(*
  Mark camera system on WEU machine
  1 mark sensor (optional: reverse mode - roll printed in reversed direction, sensor moved to other side)
*)
FUNCTION_BLOCK FB_MarkCamera_WEU EXTENDS FB_CameraBase
VAR_INPUT
  bReadyForPrinting             : BOOL;     // 
  nCurrentPosition              : DINT;     // current print postion
  fCurrentSpeed                 : LREAL;    // current print speed
  bPrintMarkExist               : BOOL;     // [from machine] print mark existing
  bPrintDirReverse              : BOOL;     // [from machine] print substrate in reverse direction
  nUsePerRepeatInLine           : UDINT;    // [from machine] use per repeat
  fMarkSizeDefault              : LREAL;    // mark size "a" [m]
  fMarkDistRepeatToStartMark    : LREAL;    // mark distance from repeat to start mark [m]
  fMarkDistFromCenter           : LREAL;    // mark distance from center [m]
END_VAR
VAR
  fbMarkDefinition   : FB_MarkDefinition;   // mark definition instance (used by MarkDetection)
  fbMarkDetection    : FB_MarkDetection;    // StartPosTrigger, CameraTrigger and MarkDetection (Mark handler for MarkCamera)
  
  // teach info
  _bTeachOk                     : BOOL;
  _nTeachedPoints               : UDINT;
  _nDetectedMarks               : UDINT;
  
  // status
  _bTeachError                  : BOOL;     // teach was not successful
  _bImageLengthError            : BOOL;     // invalid image/repeat length
  _bMarkDefinitionError         : BOOL;     // invalid mark definition
END_VAR
VAR CONSTANT
  fC_MinImageLength : LREAL := 0.05;  // minimal "repeat" length
END_VAR
VAR PERSISTENT
  eMarkMode     : E_MarkMode := E_MarkMode.AutoDefault;   // mark generation/detection mode
  bMarkInverted : BOOL;             // mark triangle are flipped on x axis
  nUsePerRepeat : UDINT := 4;       // number of "use" per repeat
  fMarkSpec_a   : LREAL := 0.005;   // mark spec a [m] - mark width
  fMarkSpec_b   : LREAL := 0.005;   // mark spec b [m] - (optional) triangle length
  fMarkSpec_c   : LREAL := 0.005;   // mark spec c [m] - start mark distance to 0
END_VAR

IF NOT _bInitialized THEN RETURN; END_IF

// The detection work is done in FB_MarkDetection
// This FB just uses(receives) the marks from the external implementation
// - Receives events CamTrigger & CamTriggerDone from MarkDetection
// - Get current marks and send them to the iCameraSink
fbMarkDetection.bSimEnable := _bSimulate;
IF _bSimulate THEN sim_update(); END_IF

fbMarkDetection(
  bEnable:=bReadyForPrinting,
  bAutomaticMode:=TRUE,
  nCurrentPos:=nCurrentPosition,
  fCurrentSpeed:=fCurrentSpeed
);

_bTeachOk := (fbMarkDefinition.nMarks > 0);
_nTeachedPoints := fbMarkDefinition.nMarks;
_nDetectedMarks := fbMarkDefinition.nMarksDetected;

IF nUsePerRepeatInLine <> nUsePerRepeat THEN nUsePerRepeat := nUsePerRepeatInLine; END_IF

IF _bCamTriggerStarted THEN sendCamPoints(); END_IF

fbMarkDefinition.update_view();

METHOD ackErrors
VAR_INPUT
END_VAR
_bTeachError := FALSE;
_bImageLengthError := FALSE;
_bMarkDefinitionError := FALSE;

fbMarkDetection.ackErrors();
END_METHOD

PROPERTY bImageLengthInvalid : BOOL
GET
bImageLengthInvalid := _bImageLengthError;
END_GET
END_PROPERTY

PROPERTY bMarkDetectionErrors : BOOL
GET
bMarkDetectionErrors := fbMarkDetection._bMarkDetectionErrors;
END_GET
END_PROPERTY

PROPERTY bMissingMarks : BOOL
GET
bMissingMarks := fbMarkDetection._bMissingMarks;
END_GET
END_PROPERTY

PROPERTY bTeachError : BOOL
GET
bTeachError := _bTeachError;
END_GET
END_PROPERTY

METHOD CamTriggerDone
IF NOT _bInitialized THEN RETURN; END_IF

// stream lasting points to Worker Camera
IF _bCamTriggerStarted THEN
  sendCamPoints();
  _iCameraSink.fPrintLengthEffective := fbMarkDetection.fEffectiveImageLength;
END_IF

SUPER^.CamTriggerDone();
END_METHOD

{attribute 'monitoring':='call'}
PROPERTY eCameraMode : E_CameraMode
GET
eCameraMode := _eCameraMode;
IF _eCameraMode = E_CameraMode.Auto THEN
  eCameraMode := E_CameraMode.Live;
END_IF
END_GET
END_PROPERTY

PROPERTY eDeviceType : E_CameraDevice
GET
eDeviceType := E_CameraDevice.PrintMark;
END_GET
END_PROPERTY

METHOD GetCamStatus : BOOL
VAR_OUTPUT
  bConnectionOK  : BOOL;    // Camera connected
  bTeachOk       : BOOL;    // Teach successful
  nTeachedPoints : UDINT;   // Teached points for this job
  nScannedPoints : UDINT;   // Scanned points on current sheet
  bCamStarted    : BOOL;    // Camera trigger is active, cam started
  bCamDone       : BOOL;    // Camera finished on last CT
  bErrors        : ARRAY[1..GVL_Camera.nC_NbCamErrors] OF BOOL;  // generic error flag list
END_VAR
bConnectionOK  := TRUE;
bTeachOk       := _bTeachOk;
nTeachedPoints := _nTeachedPoints;
nScannedPoints := _nRxCamPoints;
bCamStarted    := _bCamTriggerStarted;
bCamDone       := _bCamTriggerDone;

GetCamStatus := bConnectionOK AND bTeachOk;   // camera ready
END_METHOD

METHOD InitMarkCamera
VAR_INPUT
  fPrintUnitResolution         : LREAL;    (*printhead pixel resolution [dpi]*)
  fPrintUnitSubPx              : LREAL;    (*print unit subPixel resolution [SubPx]*)
END_VAR
VAR
  bOK : BOOL;
END_VAR
SUPER^.Init( 
  nPrintUnitResolution      := TO_UDINT(fPrintUnitResolution),
  nPrintUnitSubPx           := TO_UDINT(fPrintUnitSubPx), 
  iCameraTrigger            := fbMarkDetection, 
  bUseCameraTrigger         := FALSE, 
  bUseCameraTriggerFeedback := FALSE
);


IF NOT _bInitialized THEN LogError('Init: invalid parameter'); RETURN; END_IF

// -- Mark definition handler
fbMarkDefinition.Init();

// -- Mark detection handler
fbMarkDetection.Init(
  fPrintResolution:=fPrintUnitResolution, 
  fSubPxResolution:=fPrintUnitSubPx, 
  pFbMarkDefinition:=ADR(fbMarkDefinition)
);

_bInitialized := TRUE;
END_METHOD

METHOD mJobStart : BOOL
// parameter checks
IF fImageLength < fC_MinImageLength THEN _bImageLengthError:=TRUE; LogError('JobStart: Repeat length (ImageLength) too small'); END_IF

// mark mode selection based on machine configuration
// No marks => None
// With marks => use AutoDefault or the special mark selected prior in ui
IF NOT bPrintMarkExist THEN 
  LogLvl(Lvl:=E_LogSeverity.Detail, Msg:='JobStart: No Marks exist, use None/Sim mode');
  eMarkMode := E_MarkMode.None;
ELSE
  IF eMarkMode = E_MarkMode.None THEN 
    eMarkMode := E_MarkMode.AutoDefault; 
  END_IF
END_IF

// get mark definition
fMarkSpec_a := fMarkSizeDefault;
fMarkSpec_c := fMarkDistRepeatToStartMark;
//fMarkSpec_b := ;

IF fMarkSpec_a = 0 THEN _bMarkDefinitionError := TRUE; LogError(F_Concat2('JobStart: MarkLength invalid "a"=', TO_STRING(fMarkSpec_a))); END_IF
IF eMarkMode = E_MarkMode.OneTriangle AND fMarkSpec_b = 0 THEN _bMarkDefinitionError := TRUE; LogError(F_Concat2('JobStart: MarkLength invalid "c"=', TO_STRING(fMarkSpec_c))); END_IF

// Teach marks based on job and configuration
IF eCameraMode <> E_CameraMode.NoCorrection THEN
  _bTeachError := NOT fbMarkDefinition.TeachMarks(
    fImageLength:=fImageLength, 
    fImageWidth:=fImageWidth, 
    eMarkMode:=eMarkMode,
    a:=fMarkSpec_a,
    b:=fMarkSpec_b,
    c:=fMarkSpec_c,
    nUses:=nUsePerRepeat,
    bMarkInverted:=bMarkInverted
  );
END_IF
END_METHOD

PROPERTY pFbMarkDefinition : POINTER TO FB_MarkDefinition
GET
pFbMarkDefinition := ADR(fbMarkDefinition);
END_GET
END_PROPERTY

// stream already detected cam points to sink.
METHOD PRIVATE sendCamPoints
VAR
  i : UDINT;
  pMark : POINTER TO ST_MarkDefinition;
END_VAR
WHILE _nRxCamPoints < fbMarkDefinition.nMarksDetected DO
  
  pMark := fbMarkDefinition.getMark(nIdx:=TO_DINT(_nRxCamPoints+1));
  IF pMark <> 0 THEN
    // Send Mark (CamPoint) to CameraSink
    stCamPoint.x_ref := F_MeterToSubPixelReal(  fPosMeter:=pMark^.fPosX                                 (*[m]*)
                                              , fResoSubPx:=UDINT_TO_LREAL(_nPrintUnitResolution));     (*Result should be in pixels*)
    stCamPoint.y_ref := F_MeterToSubPixelReal( fPosMeter:=pMark^.fPosY                                  (*[m]*)
                                              , fResoSubPx:=UDINT_TO_LREAL(_nPrintUnitResolution));     (*Result should be in pixels*)
    stCamPoint.dx    := F_MeterToSubPixelReal( fPosMeter:=pMark^.sState.dx                              (*[m]*)
                                              , fResoSubPx:=UDINT_TO_LREAL(_nPrintUnitResolution));     (*Result should be in pixels*)
    stCamPoint.dy    := F_MeterToSubPixelReal( fPosMeter:=pMark^.sState.dy                              (*[m]*)
                                              , fResoSubPx:=UDINT_TO_LREAL(_nPrintUnitResolution));     (*Result should be in pixels*)
    stCamPoint.valid := pMark^.sState.bSet;
  
    IF _iCameraSink <> 0 THEN
      _iCameraSink.AddCamPoint(sDeformationPoint:=stCamPoint);
    END_IF
  ELSE
    LogWarning(F_Concat2('Requested mark not found, mark Idx=', TO_STRING(_nRxCamPoints+1)));
  END_IF
  
  _nRxCamPoints := _nRxCamPoints + 1;   // next mark
END_WHILE
END_METHOD

(*
  Set mode to camera.
  :return: TRUE if success
*)
METHOD setCameraMode : BOOL
VAR_INPUT
  eCameraMode : E_CameraMode;
END_VAR
IF eCameraMode = E_CameraMode.Auto OR
   eCameraMode = E_CameraMode.NoCorrection OR
   eCameraMode = E_CameraMode.Live
   //eCameraMode = E_CameraMode.Trend 
THEN
   
  _eCameraMode := eCameraMode;  // set desired mode
  setCameraMode := TRUE;
ELSE
  LogError(F_Concat3('Camera mode=', TO_STRING(eCameraMode), ' not supported by camera'));
  _eCameraMode := E_CameraMode.NoCorrection;
END_IF
END_METHOD

METHOD PRIVATE sim_update
// nothing
END_METHOD

{attribute 'monitoring':='variable'}
PROPERTY sName : STRING
GET
sName := 'Printmarks';
END_GET
END_PROPERTY

END_FUNCTION_BLOCK

(* stored: Version 1.1.0.1, ProductVersion 3.1.4024.11
   POU FB_MarkCamera_WEU: Id {afee498a-a574-4419-ba71-cf35979d8699}, SpecialFunc None
   Folder Errors: Id {a01e90ed-adf1-4c3e-a3f6-2cabd0d609d0}
   Folder I_CameraTriggerDevice: Id {4773bc35-df63-4cfd-9fcd-8027e8678bf9}
   Method ackErrors: Id {6d381463-10c6-4dda-a89c-e8be47d736f9}
   Property bImageLengthInvalid: Id {8ce60234-4f56-4d8f-b2aa-0e2e0adae3b0}
   Get Get: Id {ca2b44a6-2f71-42bc-8246-d8f9916a6bd7}
   Property bMarkDetectionErrors: Id {7a1a4e25-3606-442c-80f7-39054a32690e}
   Get Get: Id {bf74de13-e67d-409d-a425-e80bf20f310d}
   Property bMissingMarks: Id {16c4d983-afb9-47fc-b3a0-43e8b8f856f1}
   Get Get: Id {bfdb3c45-61da-45e4-90ca-803c164e5fdf}
   Property bTeachError: Id {d32145c6-71bd-404c-9468-3a12da2d9f73}
   Get Get: Id {b090c8ba-d759-47b7-a0ca-23e6705d2988}
   Method CamTriggerDone: Id {d41794c6-1f76-436d-8466-03ff8773ac59}
   Property eCameraMode: Id {b022aee1-cf4c-4fcc-81a5-0dbe1bef2090}
   Get Get: Id {bf30cebf-f837-493d-a842-a0d56f30c0ad}
   Property eDeviceType: Id {84e5cd81-ce1f-4baf-9ea0-b8044b8893cd}
   Get Get: Id {63d06dd5-4d22-4f3f-a574-84fddd78ad77}
   Method GetCamStatus: Id {38e7ce1d-c905-4dcd-bcee-13c392fb6b4e}
   Method InitMarkCamera: Id {51f51649-6984-44e8-9e66-86e2adb32565}
   Method mJobStart: Id {eb0884e6-0b51-420a-ab81-2fa58f38387d}
   Property pFbMarkDefinition: Id {7c064055-0d1a-4195-ad1f-3f4c34609c08}
   Get Get: Id {6e9035d1-f48d-4704-82b2-6002f7c8f9a3}
   Method sendCamPoints: Id {79d0c237-9754-4336-866d-7de126f506b7}
   Method setCameraMode: Id {54a34304-23e4-4c00-9f45-c8cea9937ff8}
   Method sim_update: Id {63e89f21-21b3-46ae-aa39-a62ec4b9499b}
   Property sName: Id {26af1a37-4820-4145-8569-298bb52be617}
   Get Get: Id {7cd4e3ff-8058-40ee-b02a-2b43197c6b96} *)
